TYPE ST_UIStatus :
STRUCT
	ComponentStatus : REFERENCE TO ST_ComponentStatus;
	ConnectionStatus	: BOOL;
END_STRUCT
END_TYPE

(* stored: Version 1.1.0.1
   DUT ST_UIStatus: Id {8010ae4a-d7a3-49e7-98fa-6b18ba4c6504} *)
